FUNCTION_BLOCK AX_NOT_INIT (* standard boolean NOT function *)
  (* Standard: 61131-3; Classification: standard boolean function; Description: Copyright (c) 2011 TU Wien ACIN, HR Agrartechnik GmbH This program and the accompanying materials are made available under the terms of the Eclipse Public License 2.0 which is available at https://www.eclipse.org/legal/epl-2.0/ SPDX-License-Identifier: EPL-2.0 *)
  (* Version 3.1, 2025-11-04, Franz Höpfinger, HR Agrartechnik GmbH, made AX Version *)
  (* Version 3.0, 2025-04-14, Patrick Aigner, changed package *)
  (* Version 1.0, 2011-06-21, Monika Wenger, TU Wien ACIN *)
  PACKAGE adapter::booleanOperators;
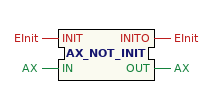
  EVENT_INPUT
    INIT : EInit; (* Initialization Request *)
  END_EVENT
  EVENT_OUTPUT
    INITO : EInit; (* Initialization Confirm *)
  END_EVENT
  SOCKETS
    IN : adapter::types::unidirectional::AX; (* Input *)
  END_SOCKETS
  PLUGS
    OUT : adapter::types::unidirectional::AX; (* Output *)
  END_PLUGS
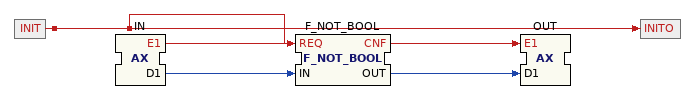
  FBS
    F_NOT_BOOL : iec61131::bitwiseOperators::F_NOT_BOOL;
  END_FBS
  EVENT_CONNECTIONS
    F_NOT_BOOL.CNF TO OUT.E1;
    IN.E1 TO F_NOT_BOOL.REQ;
    INIT TO INITO;
    INIT TO F_NOT_BOOL.REQ;
  END_CONNECTIONS
  DATA_CONNECTIONS
    F_NOT_BOOL.OUT TO OUT.D1;
    IN.D1 TO F_NOT_BOOL.IN;
  END_CONNECTIONS
END_FUNCTION_BLOCK
